// TIA Portal project "DemoProject_V17" (V17)

(* hardware
DEVICE "S71500/ET200MP station_1"  S7-1500 station
   slot 0: "Rail_0"  Rack  6ES7 590-1***0-0AA0
   slot 1: "PLC_1"  CPU 1518-4 PN/DP  6ES7 518-4AP00-0AB0  V2.6
      slot 3: "CPU display_1"  6ES7591-1BA00-0AA0
      slot 32768: "PROFINET interface_1"  X1
         slot 32769: "Port_1"  X1 P1
         slot 32770: "Port_2"  X1 P2
      slot 33024: "PROFINET interface_2"  X2
         slot 33025: "Port_1"  X2 P1
      slot 33280: "PROFINET interface GBIT_3"  X3
         slot 33281: "Port_1"  X3 P1
      slot 33536: "DP interface_1"  X4
   slot 2: "AI 4xU/I/RTD/TC / AQ 2xU/I ST_1"  AI/AQ 4xU/I/RTD/TC / 2xU/I ST  6ES7 534-7QE00-0AB0  V1.0
*)

// ===== PLC "PLC_1"  CPU 1518-4 PN/DP =====

VAR_GLOBAL   // PLC tag table "Default tag table"
   "Side A" AT %IW0 : Int;
   "Side B" AT %IW2 : Int;
   "Hypotneus(1)" AT %QW0 : Int;
END_VAR

DATA_BLOCK "Pythagoras_DB"   // DB1
{ S7_Optimized_Access := 'TRUE' }
VERSION : 0.1
// stored: InstanceOfName Pythagoras
"Pythagoras"
BEGIN
END_DATA_BLOCK

// folder: testEnvironment

DATA_BLOCK "InstPythagoras"   // DB2
{ S7_Optimized_Access := 'TRUE' }
VERSION : 0.1
// stored: InstanceOfName Pythagoras
"Pythagoras"
BEGIN
END_DATA_BLOCK

// folder: (top level)

FUNCTION_BLOCK "Pythagoras"   // FB1, SCL
{ S7_Optimized_Access := 'TRUE' }
VERSION : 0.1
   VAR_INPUT
      "a" : Real;
      "b" : Real;
   END_VAR
   VAR_OUTPUT
      valid : Bool;
      c : Real;
   END_VAR
BEGIN
   // Pythagoras formula
   // a^2 + b^2 = c^2

   IF (#a >= 0.0 AND #b >= 0.0) THEN
       #valid := true;
       #c := SQRT_REAL(#a * #a + #b * #b);
   ELSE
       #valid := false;
       #c := -1.0;
   END_IF;
END_FUNCTION_BLOCK

ORGANIZATION_BLOCK "Main"   // OB1, LAD, ProgramCycle
TITLE = "Main Program Sweep (Cycle)"
{ S7_Optimized_Access := 'TRUE' }
VERSION : 0.1
   VAR_INPUT
      Initial_Call : Bool;   // Initial call of this OB
      Remanence : Bool;   // =True, if remanent data are available
   END_VAR
BEGIN

REGION Network 1
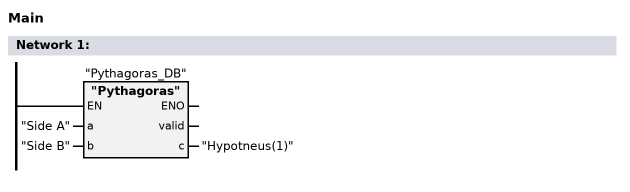
   RUNG wire#powerrail
      "Pythagoras_DB"("a" := "Side A", "b" := "Side B", valid =>, c => "Hypotneus(1)")
   END_RUNG
   // the same network as SCL:
   "Pythagoras_DB"("a" := "Side A", "b" := "Side B", c => "Hypotneus(1)");   // "Pythagoras"
END_REGION
END_ORGANIZATION_BLOCK

// folder: testEnvironment

ORGANIZATION_BLOCK "Test"   // OB123, SCL, ProgramCycle
TITLE = "Main Program Sweep (Cycle)"
{ S7_Optimized_Access := 'TRUE' }
VERSION : 0.1
   VAR_INPUT
      Initial_Call : Bool;   // Initial call of this OB
      Remanence : Bool;   // =True, if remanent data are available
   END_VAR
BEGIN
   // Test calls without parameters
   "InstPythagoras"();
END_ORGANIZATION_BLOCK